// TwinCAT 3 PLC project PLC
// ProgramVersion: 3.1.4023.0
// libraries:
//   Tc2_Standard, * (Beckhoff Automation GmbH)
//   Tc2_System, * (Beckhoff Automation GmbH)
//   Tc2_Utilities, * (Beckhoff Automation GmbH)
//   Tc3_Module, * (Beckhoff Automation GmbH)
// project tree:
//   / PlcTask.TcTTO
//   POUs/ FB_FileIO.TcPOU, MAIN.TcPOU
// real-time tasks:
//   TASK PlcTask: cycle T#10ms, priority 20, ADS port 350

CONFIGURATION PLC
    RESOURCE PLC ON TwinCAT3
        TASK PlcTask(INTERVAL := T#10ms, PRIORITY := 20);
        PROGRAM MAIN WITH PlcTask : MAIN;
    END_RESOURCE
END_CONFIGURATION

// ---- POUs/MAIN.TcPOU
PROGRAM MAIN
VAR
	fbFileIO 		: FB_FileIO;
	
	sReadPath		: STRING := 'C:\TestFile.txt';
	sWritePath		: STRING := 'C:\TestFile.txt';
	sCopyPath		: STRING := 'C:\TestCopy.txt';
	
	sTestRead		: STRING(255);
	arReadData		: ARRAY[0..255] OF BYTE;
	
	sTestWrite		: STRING(255);
	sTestAppend		: STRING;
	
	sReadArray		: ARRAY[0..9] OF T_MaxString;
	sWriteArray		: ARRAY[0..9] OF T_MaxString;
	
	sException		: STRING;
	
	i				: DINT;
	bFileExists		: BOOL;
	iFileSize		: DINT;
	
	bWriteAllText: BOOL;
	bAppendText: BOOL;
	bAppendLines: BOOL;
	bWriteAllLines: BOOL;
	bWriteAllBytes: BOOL;
	bReadAllText: BOOL;
	bReadAllLines: BOOL;
	bReadAllBytes: BOOL;
	bCheckExists: BOOL;
	bCopyFile: BOOL;
	bDeleteFile: BOOL;
	bReadSize: BOOL;
	
END_VAR

// cyclic FB call - no longer needed
//fbFileIO();

// copy exception info
sException := fbFileIO.Exception;

/// File Writes

IF bWriteAllText THEN
	sTestWrite := 'Write this string to a file. $N';
	
	// Write Text
	IF fbFileIO.WriteAllText(sWritePath, sTestWrite) THEN
		bWriteAllText := FALSE;
	END_IF
END_IF

IF bAppendText THEN
	sTestWrite := 'Append this string to a file. $N';
	
	// Append Text
	IF fbFileIO.AppendText(sWritePath, sTestWrite) THEN
		bAppendText := FALSE;
	END_IF
END_IF

IF bAppendLines THEN
	FOR i := 0 TO 4 DO
		sWriteArray[i] := CONCAT('$0AAppended Line ', TO_STRING(i));
	END_FOR
	
	// Append Lines
	IF fbFileIO.AppendLines(sWritePath, FALSE, sWriteArray) THEN
		bAppendLines := FALSE;
	END_IF
END_IF

IF bWriteAllLines THEN
	FOR i := 0 TO 4 DO
		sWriteArray[i] := CONCAT('Overwrite contents line ', TO_STRING(i));
	END_FOR
	
	// Write Lines from Array
	IF fbFileIO.WriteAllLines(sWritePath, TRUE, sWriteArray) THEN
		bWriteAllLines := FALSE;
	END_IF
END_IF

IF bWriteAllBytes THEN
	
	// Write Binary Data
	IF fbFileIO.WriteAllBytes(sCopyPath, arReadData) THEN
		bWriteAllBytes := FALSE;
	END_IF
END_IF

/// Read tests

IF bReadAllText THEN
	
	// Read Text
	IF fbFileIO.ReadAllText(sReadPath, sTestRead) THEN
		bReadAllText := FALSE;
	END_IF
END_IF

IF bReadAllLines THEN
	
	// Read Lines to Array
	IF fbFileIO.ReadAllLines(sReadPath, sReadArray) THEN
		bReadAllLines := FALSE;
	END_IF
END_IF

IF bReadAllBytes THEN
	
	// Read Binary Data
	IF fbFileIO.ReadAllBytes(sReadPath, arReadData) THEN
		bReadAllBytes := FALSE;
	END_IF
END_IF

/// File Operations

IF bCheckExists THEN
	
	// Check if File Exists (sync method - can be called inline)
	bFileExists := fbFileIO.Exists(sCopyPath);
	bCheckExists := FALSE;
END_IF

IF bCopyFile THEN
	
	// Copy File
	IF fbFileIO.CopyFile(sWritePath, sCopyPath) THEN
		bCopyFile := FALSE;
	END_IF
END_IF

IF bDeleteFile THEN
	
	// Delete File
	IF fbFileIO.DeleteFile(sCopyPath) THEN
		bDeleteFile := FALSE;
	END_IF
END_IF

IF bReadSize THEN
	
	IF fbFileIO.GetSize(sWritePath, iFileSize) THEN
		bReadSize := FALSE;
	END_IF
END_IF

END_PROGRAM

// ---- POUs/FB_FileIO.TcPOU
{attribute 'hide_all_locals'}
FUNCTION_BLOCK FB_FileIO
VAR
	// open / close FBs
	_fbFileOpen			: FB_FileOpen;
	_fbFileClose		: FB_FileClose;
	
	// reader FBs
	_fbFileRead 		: FB_FileRead;
	_fbLineRead			: FB_FileGets;
	
	// seek/tell
	_fbSeek				: FB_FileSeek;
	_fbTell				: FB_FileTell;
	
	// writer FBs
	_fbFileWrite 		: FB_FileWrite;
	_fbLineWrite		: FB_FilePuts;
	_fbFileDelete		: FB_FileDelete;
	
	// shared locals
	_nHandle			: UINT;
	_nSeq				: DINT;
	_nIdx				: DINT;
	
	_copyBuffer			: POINTER TO BYTE;
	_copyRW				: BOOL;
	
	// property fields w/ init values
	_nMaxReadLen		: DINT := 1048576;
	_tReadTimeout		: TIME := T#1S;
	
	_nMaxWriteLen		: DINT := 1048576;
	_tWriteTimeout		: TIME := T#1S;
	_bTrimWriteData		: BOOL := TRUE;
	
	_sException			: STRING;
END_VAR

// cyclic calls
THIS^.Execute();

// Appends a string array to a file. If the file does not exist, it is created.
METHOD AppendLines : BOOL
VAR_INPUT
	// Path of file to write
	Path			: STRING;
	// Insert Newlines chars after each array element
	InsertNewlines	: BOOL;
END_VAR
VAR_IN_OUT
	// Array of strings to write
	Contents		: ARRAY[*] OF T_MaxString;
END_VAR
VAR
	_sMeth			: STRING := 'AppendLines(): ';
	_sLine			: T_MaxString;
END_VAR
CASE _nSeq OF
	0 : 
		_sException := '';
		_nHandle := 0;
		
		_fbFileOpen(sPathName := Path, nMode := (FOPEN_MODETEXT OR FOPEN_MODEAPPEND), bExecute := TRUE);
		_nSeq := 1;
		
	1 :
		IF NOT _fbFileOpen.bBusy THEN
			_fbFileOpen(bExecute := FALSE);
			IF _fbFileOpen.bError THEN
				_sException := 'Error in FB_FileOpen; ';
				_sException := CONCAT(_sException, TO_STRING(_fbFileOpen.nErrId));
				_nSeq := 9;
			ELSE
				_nHandle := _fbFileOpen.hFile;
				_nIdx := LOWER_BOUND(Contents, 1);
				_nSeq := 2;
			END_IF
		END_IF
		
	2 :
		IF (_nIdx <= UPPER_BOUND(Contents, 1)) THEN
			IF Contents[_nIdx] <> '' THEN
				_sLine := SEL(InsertNewlines, Contents[_nIdx], CONCAT(Contents[_nIdx], '$0A'));
				_fbLineWrite(hFile := _nHandle, sLine := _sLine, 
					tTimeout := _tWriteTimeout, bExecute := TRUE);
			END_IF
			_nSeq := 3;
		ELSE
			_nSeq := 4;
		END_IF
		
	3 :
		IF NOT _fbLineWrite.bBusy THEN
			_fbLineWrite(bExecute := FALSE);
			IF _fbLineWrite.bError THEN
				_sException := 'Error in FB_FilePuts; ';
				_sException := CONCAT(_sException, TO_STRING(_fbLineWrite.nErrId));
				_nSeq := 9;
			ELSE
				_nIdx := _nIdx + 1;
				_nSeq := 2;
			END_IF
		END_IF
		
	
	4 : 
		_fbFileClose(hFile := _nHandle, bExecute := TRUE);
		_nSeq := 5;
		
	5 : 
		IF NOT _fbFileClose.bBusy THEN
			_fbFileClose(bExecute := FALSE);
			IF _fbFileClose.bError THEN
				_sException := 'Error in FB_FileClose; ';
				_sException := CONCAT(_sException, TO_STRING(_fbFileClose.nErrId));
				_nHandle := 0;
				_nSeq := 9;
			ELSE
				_nSeq := 0;
				AppendLines := TRUE;
			END_IF
		END_IF
		
	9 : 
		IF _nHandle <> 0 THEN
			_nSeq := 4;
		ELSE
			_sException := CONCAT(_sMeth, _sException);
			
			_nSeq := 0;
			AppendLines := TRUE;
		END_IF
		
END_CASE

THIS^.Execute();

RETURN;
END_METHOD

// Appends a string to a file. If the file does not exist, it is created.
METHOD AppendText : BOOL
VAR_INPUT
	// Path of file to append write string
	Path			: STRING;
	// String to append
	Contents		: ANY;
END_VAR
VAR
	_sMeth			: STRING := 'AppendText(): ';
	_nWriteLen		: DINT;
	_pCharIdx		: POINTER TO BYTE;
	_charVal		: BYTE;
END_VAR
IF UDINT_TO_INT(Contents.TypeClass) <> 16 THEN
	_sException := 'WriteData parameter is invalid type (STRING).';
	AppendText := TRUE;
END_IF

CASE _nSeq OF
	0 : 
		_sException := '';
		_nHandle := 0;
		
		_fbFileOpen(sPathName := Path, nMode := (FOPEN_MODETEXT OR FOPEN_MODEAPPEND), bExecute := TRUE);
		_nSeq := 1;
		
	1 :
		IF NOT _fbFileOpen.bBusy THEN
			_fbFileOpen(bExecute := FALSE);
			IF _fbFileOpen.bError THEN
				_sException := 'Error in FB_FileOpen; ';
				_sException := CONCAT(_sException, TO_STRING(_fbFileOpen.nErrId));
				_nSeq := 9;
			ELSE
				_nHandle := _fbFileOpen.hFile;
				_nSeq := 2;
			END_IF
		END_IF
		
	2 :
		IF _bTrimWriteData THEN
			_nWriteLen := THIS^.TrimLen(Contents.pValue, Contents.diSize);
		ELSE
			_nWriteLen := SEL((Contents.diSize > _nMaxWriteLen), Contents.diSize, _nMaxWriteLen);
		END_IF
		
		_fbFileWrite(hFile := _nHandle, pWriteBuff := Contents.pValue, cbWritelen := TO_UDINT(_nWriteLen), 
			tTimeout := _tWriteTimeout, bExecute := TRUE);
			
		_nSeq := 3;
		
	3 :
		IF NOT _fbFileWrite.bBusy THEN
			_fbFileWrite(bExecute := FALSE);
			IF _fbFileWrite.bError THEN
				_sException := 'Error in FB_FileWrite; ';
				_sException := CONCAT(_sException, TO_STRING(_fbFileWrite.nErrId));
				_nSeq := 9;
			ELSE
				_nSeq := 4;
			END_IF
		END_IF
		
	
	4 : 
		_fbFileClose(hFile := _nHandle, bExecute := TRUE);
		_nSeq := 5;
		
	5 : 
		IF NOT _fbFileClose.bBusy THEN
			_fbFileClose(bExecute := FALSE);
			IF _fbFileClose.bError THEN
				_sException := 'Error in FB_FileClose; ';
				_sException := CONCAT(_sException, TO_STRING(_fbFileClose.nErrId));
				_nHandle := 0;
				_nSeq := 9;
			ELSE
				_nSeq := 0;
				AppendText := TRUE;
			END_IF
		END_IF
		
	9 : 
		IF _nHandle <> 0 THEN
			_nSeq := 4;
		ELSE
			_sException := CONCAT(_sMeth, _sException);
			
			_nSeq := 0;
			AppendText := TRUE;
		END_IF
		
END_CASE

THIS^.Execute();

RETURN;
END_METHOD

// Creates a copy of the source file
METHOD CopyFile : BOOL
VAR_INPUT
	// Path of source file
	Source			: STRING;
	// Path of destination file
	Destination		: STRING;
END_VAR
VAR
	_sMeth			: STRING := 'CopyFile(): ';
	_nReadLen		: UDINT;
END_VAR

CASE _nSeq OF
	0 :
		_sException := '';
		_copyRW := FALSE;
		_nSeq := 1;
		
	1 : 
		_nHandle := 0;
		
		IF NOT _copyRW THEN
			_fbFileOpen(sPathName := Source, nMode := (FOPEN_MODEBINARY OR FOPEN_MODEREAD), bExecute := TRUE);
		ELSE
			_fbFileOpen(sPathName := Destination, nMode := (FOPEN_MODEBINARY OR FOPEN_MODEWRITE), bExecute := TRUE);
		END_IF
		
		_nSeq := 2;
		
	2 :
		IF NOT _fbFileOpen.bBusy THEN
			_fbFileOpen(bExecute := FALSE);
			IF _fbFileOpen.bError THEN
				_sException := 'Error in FB_FileOpen; ';
				_sException := CONCAT(_sException, TO_STRING(_fbFileOpen.nErrId));
				_nSeq := 9;
			ELSE
				_nHandle := _fbFileOpen.hFile;
				_nSeq := SEL(_copyRW, 3, 5);
			END_IF
		END_IF
		
	3 : 
		_copyBuffer := __NEW(BYTE, TO_UDINT(_nMaxReadLen));
		_fbFileRead(hFile := _nHandle, pReadBuff := _copyBuffer, 
			cbReadLen := TO_UDINT(_nMaxReadLen), tTimeout := _tReadTimeout, bExecute := TRUE);
			
		_nSeq := 4;
		
	4 :
		IF (NOT _fbFileRead.bBusy) OR _fbFileRead.bEOF THEN
			_fbFileRead(bExecute := FALSE);
			IF _fbFileRead.bError THEN
				_sException := 'Error in FB_FileRead; ';
				_sException := CONCAT(_sException, TO_STRING(_fbFileRead.nErrId));
				_nSeq := 9;
			ELSE
				_nSeq := 7;
			END_IF
		END_IF
		
	5 : 
		_nReadLen := _fbFileRead.cbRead;
		
		_fbFileWrite(hFile := _nHandle, pWriteBuff := _copyBuffer, cbWritelen := _nReadLen, 
			tTimeout := _tWriteTimeout, bExecute := TRUE);
			
		_nSeq := 6;
		
	6 : 
		IF NOT _fbFileWrite.bBusy THEN
			_fbFileWrite(bExecute := FALSE);
			__DELETE(_copyBuffer);
			IF _fbFileWrite.bError THEN
				_sException := 'Error in FB_FileWrite; ';
				_sException := CONCAT(_sException, TO_STRING(_fbFileWrite.nErrId));
				_nSeq := 9;
			ELSE
				_nSeq := 7;
			END_IF
		END_IF
		
		
	7 : 
		_fbFileClose(hFile := _nHandle, bExecute := TRUE);
		_nSeq := 8;
		
	8 : 
		IF NOT _fbFileClose.bBusy THEN
			_fbFileClose(bExecute := FALSE);
			IF _fbFileClose.bError THEN
				_sException := 'Error in FB_FileClose; ';
				_sException := CONCAT(_sException, TO_STRING(_fbFileClose.nErrId));
				_nHandle := 0;
				_nSeq := 9;
			ELSE
				IF _copyRW THEN
					_nSeq := 0;
					CopyFile := TRUE;
				ELSE
					_copyRW := TRUE;
					_nSeq := 1;
				END_IF
			END_IF
		END_IF
		
	9 :
		IF (_copyBuffer <> 0) THEN
			__DELETE(_copyBuffer);
		END_IF
		
		IF _nHandle <> 0 THEN
			_nSeq := 7;
		ELSE
			_sException := CONCAT(_sMeth, _sException);
			_nSeq := 0;
			CopyFile := TRUE;
		END_IF
		
END_CASE

THIS^.Execute();

RETURN;
END_METHOD

// Deletes file
METHOD DeleteFile : BOOL
VAR_INPUT
	// File path
	Path			: STRING;
END_VAR
VAR
	_sMeth			: STRING := 'DeleteFile(): ';
END_VAR
CASE _nSeq OF
	0 : 
		_sException := '';
		_nHandle := 0;
		
		_fbFileDelete(sPathName := Path, tTimeout := _tWriteTimeout, bExecute := TRUE);
		_nSeq := 1;
		
	1 : 
		IF NOT _fbFileDelete.bBusy THEN
			_fbFileDelete(bExecute := FALSE);
			IF _fbFileDelete.bError THEN
				_sException := 'Error in FB_FileDelete; ';
				_sException := CONCAT(_sException, TO_STRING(_fbFileDelete.nErrId));
				_nSeq := 9;
			ELSE
				_nSeq := 0;
				DeleteFile := TRUE;
			END_IF
		END_IF
		
	9 : 
		_sException := CONCAT(_sMeth, _sException);
		
		_nSeq := 0;
		DeleteFile := TRUE;
		
END_CASE

THIS^.Execute();

RETURN;
END_METHOD

// Last Operation Exception String
PROPERTY Exception : STRING
GET
Exception := _sException;
END_GET
END_PROPERTY

METHOD PRIVATE Execute : BOOL
VAR_INPUT
END_VAR
/// Cyclic FB calls

// file open/close
_fbFileOpen();
_fbFileClose();

// file read
_fbFileRead();
_fbLineRead();
_fbSeek();
_fbTell();

// file write
_fbFileWrite();
_fbLineWrite();

// file delete
_fbFileDelete();
END_METHOD

// Check if file exists [Synchronous Method]
METHOD Exists : BOOL
VAR_INPUT
	// Path to file
	Path			: STRING;
END_VAR
VAR
	_sMeth			: STRING := 'Exists(): ';
	_bDone			: BOOL := FALSE;
END_VAR

WHILE NOT _bDone DO
	
	_fbFileOpen();
	_fbFileClose();
	
	CASE _nSeq OF
		0 :
			_sException := '';
			_fbFileOpen(sPathName := Path, nMode := (FOPEN_MODEBINARY OR FOPEN_MODEREAD), bExecute := TRUE);
			_nSeq := 1;
			
		1 :
			IF NOT _fbFileOpen.bBusy THEN
				_fbFileOpen(bExecute := FALSE);
				IF _fbFileOpen.bError THEN
					IF _fbFileOpen.nErrId = 16#70C THEN
						_nSeq := 0;
						_bDone := TRUE;
					ELSE
						_sException := 'Error in FB_FileOpen; ';
						_sException := CONCAT(_sException, TO_STRING(_fbFileOpen.nErrId));
						_nSeq := 9;
					END_IF
					Exists := FALSE;
				ELSE
					_nHandle := _fbFileOpen.hFile;
					_nSeq := 4;
					Exists := TRUE;
				END_IF
			END_IF
			
		4 : 
			_fbFileClose(hFile := _nHandle, bExecute := TRUE);
			_nSeq := 5;
			
		5 : 
			IF NOT _fbFileClose.bBusy THEN
				_fbFileClose(bExecute := FALSE);
				IF _fbFileClose.bError THEN
					_sException := 'Error in FB_FileClose; ';
					_sException := CONCAT(_sException, TO_STRING(_fbFileClose.nErrId));
					_nHandle := 0;
					_nSeq := 9;
				ELSE
					_nSeq := 0;
					_bDone := TRUE;
				END_IF
			END_IF
			
		9 :
			IF _nHandle <> 0 THEN
				_nSeq := 4;
			ELSE
				_sException := CONCAT(_sMeth, _sException);
				_nSeq := 0;
				_bDone := TRUE;
			END_IF
			
	END_CASE
	
END_WHILE

RETURN;
END_METHOD

// Gets the file size in bytes
METHOD GetSize : BOOL
VAR_INPUT
	// Path to file
	Path			: STRING;
	//	File size
	FileSize		: REFERENCE TO DINT;
END_VAR
VAR
	_sMeth			: STRING := 'GetSize(): ';
END_VAR

CASE _nSeq OF
	0 :
		_sException := '';
		_nHandle := 0;
		
		_fbFileOpen(sPathName := Path, nMode := (FOPEN_MODEBINARY OR FOPEN_MODEREAD), bExecute := TRUE);
		_nSeq := 1;
		
	1 :
		IF NOT _fbFileOpen.bBusy THEN
			_fbFileOpen(bExecute := FALSE);
			IF _fbFileOpen.bError THEN
				_sException := 'Error in FB_FileOpen; ';
				_sException := CONCAT(_sException, TO_STRING(_fbFileOpen.nErrId));
				_nSeq := 9;
			ELSE
				_nHandle := _fbFileOpen.hFile;
				_nSeq := 2;
			END_IF
		END_IF
		
	2 : 
		_fbSeek(sNetId := '', hFile := _nHandle, eOrigin := E_SeekOrigin.SEEK_END, bExecute := TRUE);
		_nSeq := 3;
		
	3 :
		IF (NOT _fbSeek.bBusy) THEN
			_fbSeek(bExecute := FALSE);
			IF _fbSeek.bError THEN
				_sException := 'Error in FB_FileSeek; ';
				_sException := CONCAT(_sException, TO_STRING(_fbSeek.nErrId));
				_nSeq := 9;
			ELSE
				_fbTell(sNetId := '', hFile := _nHandle, bExecute := TRUE);
				_nSeq := 4;
			END_IF
		END_IF
		
	4 : 
		IF (NOT _fbTell.bBusy) THEN
			_fbTell(bExecute := FALSE);
			IF _fbTell.bError THEN
				_sException := 'Error in FB_FileTell; ';
				_sException := CONCAT(_sException, TO_STRING(_fbTell.nErrId));
				_nSeq := 9;
			ELSE
				FileSize := _fbTell.nSeekPos;
				_nSeq := 5;
			END_IF
		END_IF
		
		
	5 : 
		_fbFileClose(hFile := _nHandle, bExecute := TRUE);
		_nSeq := 6;
		
	6 : 
		IF NOT _fbFileClose.bBusy THEN
			_fbFileClose(bExecute := FALSE);
			IF _fbFileClose.bError THEN
				_sException := 'Error in FB_FileClose; ';
				_sException := CONCAT(_sException, TO_STRING(_fbFileClose.nErrId));
				_nHandle := 0;
				_nSeq := 9;
			ELSE
				_nSeq := 0;
				GetSize := TRUE;
			END_IF
		END_IF
		
	9 :
		IF _nHandle <> 0 THEN
			_nSeq := 4;
		ELSE
			_sException := CONCAT(_sMeth, _sException);
			
			_nSeq := 0;
			GetSize := TRUE;
		END_IF
		
END_CASE

THIS^.Execute();

RETURN;
END_METHOD

// Maximum File Read Length (bytes) Default: 1048576 (1MB)
PROPERTY MaxReadLen : DINT
GET
MaxReadLen := _nMaxReadLen;
END_GET
SET
_nMaxReadLen := MaxReadLen;
END_SET
END_PROPERTY

// Maximum File Write Length (bytes) Default: 1048576 (1MB)
PROPERTY MaxWriteLen : DINT
GET
MaxWriteLen := _nMaxWriteLen;
END_GET
SET
_nMaxWriteLen := MaxWriteLen;
END_SET
END_PROPERTY

// Read the binary content of a file into an array of bytes
METHOD ReadAllBytes : BOOL
VAR_INPUT
	// Path of File to Read
	Path			: STRING;
END_VAR
VAR_IN_OUT
	// Array of bytes to store read data
	Contents		: ARRAY[*] OF BYTE;
END_VAR
VAR
	_nReadLen		: DINT;
	_sMeth			: STRING := 'ReadAllBytes(): ';
END_VAR

CASE _nSeq OF
	0 :
		_sException := '';
		_nHandle := 0;
		
		_fbFileOpen(sPathName := Path, nMode := (FOPEN_MODEBINARY OR FOPEN_MODEREAD), bExecute := TRUE);
		_nSeq := 1;
		
	1 :
		IF NOT _fbFileOpen.bBusy THEN
			_fbFileOpen(bExecute := FALSE);
			IF _fbFileOpen.bError THEN
				_sException := 'Error in FB_FileOpen; ';
				_sException := CONCAT(_sException, TO_STRING(_fbFileOpen.nErrId));
				_nSeq := 9;
			ELSE
				_nHandle := _fbFileOpen.hFile;
				_nSeq := 2;
			END_IF
		END_IF
		
	2 : 
		_nReadLen := UPPER_BOUND(Contents, 1) - LOWER_BOUND(Contents, 1) + 1;
		MEMSET(Contents, 0, TO_UDINT(_nReadLen));
		_nReadLen := SEL((_nReadLen > _nMaxReadLen), _nReadLen, _nMaxReadLen);
		
		_fbFileRead(hFile := _nHandle, pReadBuff := Contents, 
			cbReadLen := TO_UDINT(_nReadLen), tTimeout := _tReadTimeout, bExecute := TRUE);
			
		_nSeq := 3;
		
	3 :
		IF (NOT _fbFileRead.bBusy) OR _fbFileRead.bEOF THEN
			_fbFileRead(bExecute := FALSE);
			IF _fbFileRead.bError THEN
				_sException := 'Error in FB_FileRead; ';
				_sException := CONCAT(_sException, TO_STRING(_fbFileRead.nErrId));
				_nSeq := 9;
			ELSE
				_nSeq := 4;
			END_IF
		END_IF
		
	4 : 
		_fbFileClose(hFile := _nHandle, bExecute := TRUE);
		_nSeq := 5;
		
	5 : 
		IF NOT _fbFileClose.bBusy THEN
			_fbFileClose(bExecute := FALSE);
			IF _fbFileClose.bError THEN
				_sException := 'Error in FB_FileClose; ';
				_sException := CONCAT(_sException, TO_STRING(_fbFileClose.nErrId));
				_nHandle := 0;
				_nSeq := 9;
			ELSE
				_nSeq := 0;
				ReadAllBytes := TRUE;
			END_IF
		END_IF
		
	9 :
		IF _nHandle <> 0 THEN
			_nSeq := 4;
		ELSE
			_sException := CONCAT(_sMeth, _sException);
			
			_nSeq := 0;
			ReadAllBytes := TRUE;
		END_IF
		
END_CASE

THIS^.Execute();

RETURN;
END_METHOD

// Reads all the lines in a file to an array of strings
METHOD ReadAllLines : BOOL
VAR_INPUT
	// Path of File to Read
	Path			: STRING;
END_VAR
VAR_IN_OUT
	// String Array to store Read Lines
	Contents		: ARRAY[*] OF T_MaxString;
END_VAR

VAR
	_sMeth			: STRING := 'ReadAllLines(): ';
END_VAR

CASE _nSeq OF
	0 :
		_sException := '';
		_nHandle := 0;
		
		_fbFileOpen(sPathName := Path, nMode := (FOPEN_MODETEXT OR FOPEN_MODEREAD), bExecute := TRUE);
		_nSeq := 1;
		
	1 :
		IF NOT _fbFileOpen.bBusy THEN
			_fbFileOpen(bExecute := FALSE);
			IF _fbFileOpen.bError THEN
				_sException := 'Error in FB_FileOpen; ';
				_sException := CONCAT(_sException, TO_STRING(_fbFileOpen.nErrId));
				_nSeq := 9;
			ELSE
				_nHandle := _fbFileOpen.hFile;
				_nIdx := LOWER_BOUND(Contents, 1);
				_nSeq := 2;
			END_IF
		END_IF
		
	2 : 
		IF (_nIdx <= UPPER_BOUND(Contents, 1)) THEN
			_fbLineRead(hFile := _nHandle, tTimeout := _tReadTimeout, bExecute := TRUE);
			_nSeq := 3;
		ELSE
			_nSeq := 4;
		END_IF
		
	3 :
		IF (NOT _fbLineRead.bBusy) OR _fbLineRead.bEOF THEN
			_fbLineRead(bExecute := FALSE);
			IF _fbLineRead.bError THEN
				_sException := 'Error in FB_FileGets; ';
				_sException := CONCAT(_sException, TO_STRING(_fbLineRead.nErrId));
				_nSeq := 9;
			ELSE
				IF _fbLineRead.bEOF THEN
					_nSeq := 4;
				ELSE
					Contents[_nIdx] := _fbLineRead.sLine;
					_nIdx := _nIdx + 1;
					_nSeq := 2;
				END_IF
			END_IF
		END_IF
		
		
	4 : 
		FOR _nIdx := _nIdx TO UPPER_BOUND(Contents, 1) DO
			Contents[_nIdx] := '';
		END_FOR
		
		_fbFileClose(hFile := _nHandle, bExecute := TRUE);
		_nSeq := 5;
		
	5 : 
		IF NOT _fbFileClose.bBusy THEN
			_fbFileClose(bExecute := FALSE);
			IF _fbFileClose.bError THEN
				_sException := 'Error in FB_FileClose; ';
				_sException := CONCAT(_sException, TO_STRING(_fbFileClose.nErrId));
				_nHandle := 0;
				_nSeq := 9;
			ELSE
				_nSeq := 0;
				ReadAllLines := TRUE;
			END_IF
		END_IF
		
	9 :
		IF _nHandle <> 0 THEN
			_nSeq := 4;
		ELSE
			_sException := CONCAT(_sMeth, _sException);
			Contents[LOWER_BOUND(Contents, 1)] := _sException;
			
			_nSeq := 0;
			ReadAllLines := TRUE;
		END_IF
		
END_CASE

THIS^.Execute();

RETURN;
END_METHOD

// Reads all the text from a file into a string
METHOD ReadAllText : BOOL
VAR_INPUT
	// Path of File to Read
	Path			: STRING;
	// String to store Read Data
	Contents		: ANY;
END_VAR
VAR
	_nReadLen		: DINT;
	_sMeth			: STRING := 'ReadAllText(): ';
END_VAR
IF UDINT_TO_INT(Contents.TypeClass) <> 16 THEN
	_sException := 'ReadData parameter is invalid type (STRING).';
	ReadAllText := TRUE;
END_IF

CASE _nSeq OF
	0 :
		_sException := '';
		_nHandle := 0;
		
		_fbFileOpen(sPathName := Path, nMode := (FOPEN_MODETEXT OR FOPEN_MODEREAD), bExecute := TRUE);
		_nSeq := 1;
		
	1 :
		IF NOT _fbFileOpen.bBusy THEN
			_fbFileOpen(bExecute := FALSE);
			IF _fbFileOpen.bError THEN
				_sException := 'Error in FB_FileOpen; ';
				_sException := CONCAT(_sException, TO_STRING(_fbFileOpen.nErrId));
				_nSeq := 9;
			ELSE
				_nHandle := _fbFileOpen.hFile;
				_nSeq := 2;
			END_IF
		END_IF
		
	2 : 
		MEMSET(Contents.pValue, 0, TO_UDINT(Contents.diSize));
		_nReadLen := SEL((Contents.diSize > _nMaxReadLen), Contents.diSize, _nMaxReadLen);
		_fbFileRead(hFile := _nHandle, pReadBuff := Contents.pValue, 
			cbReadLen := TO_UDINT(_nReadLen), tTimeout := _tReadTimeout, bExecute := TRUE);
			
		_nSeq := 3;
		
	3 :
		IF (NOT _fbFileRead.bBusy) OR _fbFileRead.bEOF THEN
			_fbFileRead(bExecute := FALSE);
			IF _fbFileRead.bError THEN
				_sException := 'Error in FB_FileRead; ';
				_sException := CONCAT(_sException, TO_STRING(_fbFileRead.nErrId));
				_nSeq := 9;
			ELSE
				_nSeq := 4;
			END_IF
		END_IF
		
	4 : 
		_fbFileClose(hFile := _nHandle, bExecute := TRUE);
		_nSeq := 5;
		
	5 : 
		IF NOT _fbFileClose.bBusy THEN
			_fbFileClose(bExecute := FALSE);
			IF _fbFileClose.bError THEN
				_sException := 'Error in FB_FileClose; ';
				_sException := CONCAT(_sException, TO_STRING(_fbFileClose.nErrId));
				_nHandle := 0;
				_nSeq := 9;
			ELSE
				_nSeq := 0;
				ReadAllText := TRUE;
			END_IF
		END_IF
		
	9 :
		IF _nHandle <> 0 THEN
			_nSeq := 4;
		ELSE
			_sException := CONCAT(_sMeth, _sException);
			MEMCPY(Contents.pValue, ADR(_sException), TO_UDINT(LEN(_sException)));
			
			_nSeq := 0;
			ReadAllText := TRUE;
		END_IF
		
END_CASE

THIS^.Execute();

RETURN;
END_METHOD

// File Read Operation Timeout (Default: T#1S)
PROPERTY ReadTimeout : TIME
GET
ReadTimeout := _tReadTimeout;
END_GET
SET
_tReadTimeout := ReadTimeout;
END_SET
END_PROPERTY

METHOD PRIVATE TrimLen : DINT
VAR_INPUT
	CharPtr		: POINTER TO BYTE;
	Len			: DINT;
END_VAR
VAR
	_pCharIdx		: POINTER TO BYTE;
	_charVal		: BYTE;
	_ret			: DINT;
END_VAR
_pCharIdx := CharPtr;
FOR _nIdx := 0 TO Len - 1 DO
	_charVal := _pCharIdx^;
	IF _charVal = 0 THEN
		EXIT;
	ELSE
		_ret := _ret + 1;
		_pCharIdx := _pCharIdx + 1;
	END_IF
END_FOR

TrimLen := _ret;
END_METHOD

// Trim null characters from write contents before writing/appending to file (Default: true)
PROPERTY TrimWriteData : BOOL
GET
TrimWriteData := _bTrimWriteData;
END_GET
SET
_bTrimWriteData := TrimWriteData;
END_SET
END_PROPERTY

// Write array of bytes to file
METHOD WriteAllBytes : BOOL
VAR_INPUT
	// Path to file
	Path			: STRING;
END_VAR
VAR_IN_OUT
	// Array of bytes to write
	Contents		: ARRAY[*] OF BYTE;
END_VAR
VAR
	_sMeth			: STRING := 'WriteAllBytes(): ';
	_nWriteLen		: DINT;
END_VAR

CASE _nSeq OF
	0 : 
		_sException := '';
		_nHandle := 0;
		
		_fbFileOpen(sPathName := Path, nMode := (FOPEN_MODEBINARY OR FOPEN_MODEWRITE), bExecute := TRUE);
		_nSeq := 1;
		
	1 :
		IF NOT _fbFileOpen.bBusy THEN
			_fbFileOpen(bExecute := FALSE);
			IF _fbFileOpen.bError THEN
				_sException := 'Error in FB_FileOpen; ';
				_sException := CONCAT(_sException, TO_STRING(_fbFileOpen.nErrId));
				_nSeq := 9;
			ELSE
				_nHandle := _fbFileOpen.hFile;
				_nSeq := 2;
			END_IF
		END_IF
		
	2 :
		_nWriteLen := UPPER_BOUND(Contents, 1) - LOWER_BOUND(Contents, 1) + 1;
		
		_fbFileWrite(hFile := _nHandle, pWriteBuff := Contents, cbWritelen := TO_UDINT(_nWriteLen), 
			tTimeout := _tWriteTimeout, bExecute := TRUE);
			
		_nSeq := 3;
		
	3 :
		IF NOT _fbFileWrite.bBusy THEN
			_fbFileWrite(bExecute := FALSE);
			IF _fbFileWrite.bError THEN
				_sException := 'Error in FB_FileWrite; ';
				_sException := CONCAT(_sException, TO_STRING(_fbFileWrite.nErrId));
				_nSeq := 9;
			ELSE
				_nSeq := 4;
			END_IF
		END_IF
		
	
	4 : 
		_fbFileClose(hFile := _nHandle, bExecute := TRUE);
		_nSeq := 5;
		
	5 : 
		IF NOT _fbFileClose.bBusy THEN
			_fbFileClose(bExecute := FALSE);
			IF _fbFileClose.bError THEN
				_sException := 'Error in FB_FileClose; ';
				_sException := CONCAT(_sException, TO_STRING(_fbFileClose.nErrId));
				_nHandle := 0;
				_nSeq := 9;
			ELSE
				_nSeq := 0;
				WriteAllBytes := TRUE;
			END_IF
		END_IF
		
	9 : 
		IF _nHandle <> 0 THEN
			_nSeq := 4;
		ELSE
			_sException := CONCAT(_sMeth, _sException);
			
			_nSeq := 0;
			WriteAllBytes := TRUE;
		END_IF
		
END_CASE

THIS^.Execute();

RETURN;
END_METHOD

// Writes a string array to a file. If the file does not exist, it is created. If the file does exist, its contents are overwritten.
METHOD WriteAllLines : BOOL
VAR_INPUT
	// Path of file to write
	Path			: STRING;
	// Insert Newlines chars after each array element
	InsertNewlines	: BOOL;
END_VAR
VAR_IN_OUT
	// Array of strings to write
	Contents		: ARRAY[*] OF T_MaxString;
END_VAR
VAR
	_sMeth			: STRING := 'WriteAllLines(): ';
	_sLine			: T_MaxString;
END_VAR
CASE _nSeq OF
	0 : 
		_sException := '';
		_nHandle := 0;
		
		_fbFileOpen(sPathName := Path, nMode := (FOPEN_MODETEXT OR FOPEN_MODEWRITE), bExecute := TRUE);
		_nSeq := 1;
		
	1 :
		IF NOT _fbFileOpen.bBusy THEN
			_fbFileOpen(bExecute := FALSE);
			IF _fbFileOpen.bError THEN
				_sException := 'Error in FB_FileOpen; ';
				_sException := CONCAT(_sException, TO_STRING(_fbFileOpen.nErrId));
				_nSeq := 9;
			ELSE
				_nHandle := _fbFileOpen.hFile;
				_nIdx := LOWER_BOUND(Contents, 1);
				_nSeq := 2;
			END_IF
		END_IF
		
	2 :
		IF (_nIdx <= UPPER_BOUND(Contents, 1)) THEN
			IF Contents[_nIdx] <> '' THEN
				_sLine := SEL(InsertNewlines, Contents[_nIdx], CONCAT(Contents[_nIdx], '$0A'));
				
				_fbLineWrite(hFile := _nHandle, sLine := _sLine, 
					tTimeout := _tWriteTimeout, bExecute := TRUE);
			END_IF
			_nSeq := 3;
		ELSE
			_nSeq := 4;
		END_IF
		
	3 :
		IF NOT _fbLineWrite.bBusy THEN
			_fbLineWrite(bExecute := FALSE);
			IF _fbLineWrite.bError THEN
				_sException := 'Error in FB_FilePuts; ';
				_sException := CONCAT(_sException, TO_STRING(_fbLineWrite.nErrId));
				_nSeq := 9;
			ELSE
				_nIdx := _nIdx + 1;
				_nSeq := 2;
			END_IF
		END_IF
		
	
	4 : 
		_fbFileClose(hFile := _nHandle, bExecute := TRUE);
		_nSeq := 5;
		
	5 : 
		IF NOT _fbFileClose.bBusy THEN
			_fbFileClose(bExecute := FALSE);
			IF _fbFileClose.bError THEN
				_sException := 'Error in FB_FileClose; ';
				_sException := CONCAT(_sException, TO_STRING(_fbFileClose.nErrId));
				_nHandle := 0;
				_nSeq := 9;
			ELSE
				_nSeq := 0;
				WriteAllLines := TRUE;
			END_IF
		END_IF
		
	9 : 
		IF _nHandle <> 0 THEN
			_nSeq := 4;
		ELSE
			_sException := CONCAT(_sMeth, _sException);
			
			_nSeq := 0;
			WriteAllLines := TRUE;
		END_IF
		
END_CASE

THIS^.Execute();

RETURN;
END_METHOD

// Writes a string to the file. If the file does not exist, it is created. If the file exists, its contents are overwritten.
METHOD WriteAllText : BOOL
VAR_INPUT
	// Path of file to write
	Path			: STRING;
	// String data to write
	Contents		: ANY;
END_VAR
VAR
	_sMeth			: STRING := 'WriteAllText(): ';
	_nWriteLen		: DINT;
	_pCharIdx		: POINTER TO BYTE;
	_charVal		: BYTE;
END_VAR
IF UDINT_TO_INT(Contents.TypeClass) <> 16 THEN
	_sException := 'WriteData parameter is invalid type (STRING).';
	WriteAllText := TRUE;
END_IF

CASE _nSeq OF
	0 : 
		_sException := '';
		_nHandle := 0;
		
		_fbFileOpen(sPathName := Path, nMode := (FOPEN_MODETEXT OR FOPEN_MODEWRITE), bExecute := TRUE);
		_nSeq := 1;
		
	1 :
		IF NOT _fbFileOpen.bBusy THEN
			_fbFileOpen(bExecute := FALSE);
			IF _fbFileOpen.bError THEN
				_sException := 'Error in FB_FileOpen; ';
				_sException := CONCAT(_sException, TO_STRING(_fbFileOpen.nErrId));
				_nSeq := 9;
			ELSE
				_nHandle := _fbFileOpen.hFile;
				_nSeq := 2;
			END_IF
		END_IF
		
	2 :
		IF _bTrimWriteData THEN
			_nWriteLen := THIS^.TrimLen(Contents.pValue, Contents.diSize);
		ELSE
			_nWriteLen := SEL((Contents.diSize > _nMaxWriteLen), Contents.diSize, _nMaxWriteLen);
		END_IF
		
		_fbFileWrite(hFile := _nHandle, pWriteBuff := Contents.pValue, cbWritelen := TO_UDINT(_nWriteLen), 
			tTimeout := _tWriteTimeout, bExecute := TRUE);
			
		_nSeq := 3;
		
	3 :
		IF NOT _fbFileWrite.bBusy THEN
			_fbFileWrite(bExecute := FALSE);
			IF _fbFileWrite.bError THEN
				_sException := 'Error in FB_FileWrite; ';
				_sException := CONCAT(_sException, TO_STRING(_fbFileWrite.nErrId));
				_nSeq := 9;
			ELSE
				_nSeq := 4;
			END_IF
		END_IF
		
	
	4 : 
		_fbFileClose(hFile := _nHandle, bExecute := TRUE);
		_nSeq := 5;
		
	5 : 
		IF NOT _fbFileClose.bBusy THEN
			_fbFileClose(bExecute := FALSE);
			IF _fbFileClose.bError THEN
				_sException := 'Error in FB_FileClose; ';
				_sException := CONCAT(_sException, TO_STRING(_fbFileClose.nErrId));
				_nHandle := 0;
				_nSeq := 9;
			ELSE
				_nSeq := 0;
				WriteAllText := TRUE;
			END_IF
		END_IF
		
	9 : 
		IF _nHandle <> 0 THEN
			_nSeq := 4;
		ELSE
			_sException := CONCAT(_sMeth, _sException);
			
			_nSeq := 0;
			WriteAllText := TRUE;
		END_IF
		
END_CASE

THIS^.Execute();

RETURN;
END_METHOD

// File Write Operation Timeout (Default: T#1S)
PROPERTY WriteTimeout : TIME
GET
WriteTimeout := _tWriteTimeout;
END_GET
SET
_tWriteTimeout := WriteTimeout;
END_SET
END_PROPERTY

END_FUNCTION_BLOCK
